{attribute addProperty BoxType "ELX9410-0000-0018"}
{attribute addProperty Id "Status_Us_InAT %I*Status_Us_In_D944C060810Status_Us_OutAT %I*Status_Us_Out_D944C060810WcStateAT %I*WcState_98A4DF7520.250InfoDataAT %I*InfoData_192954DE1620"}
{attribute addProperty CRC "974068585"}
{attribute addProperty SizeInBites "34"}
{attribute addProperty SizeInBytes "4.25"}
TYPE ELX9410_B5764C82 :
STRUCT
	{attribute addProperty Name "Status_Us_In"}
	Status_Us_In : Status_Us_In_D944C060;
	{attribute addProperty Name "Status_Us_Out"}
	Status_Us_Out : Status_Us_Out_D944C060;
	{attribute addProperty Name "WcState"}
	WcState : WcState_98A4DF75;
	{attribute addProperty Name "InfoData"}
	InfoData : InfoData_192954DE;
END_STRUCT
END_TYPE

(* stored: Version 1.2.0.0, ProductVersion 3.1.4024.9
   DUT ELX9410_B5764C82: Id {fad88d35-4993-491f-bd7d-0c53dd744f93} *)
